// Mitsubishi GX Works2 project: LRI - PLC - A1+Ã1+A2   PLC: Q03UDV

PROGRAM MAIN
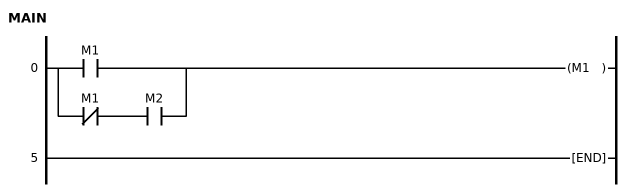
0     LD      M1
      LDI     M1
      AND     M2
      ORB
      OUT     M1
5     END
END_PROGRAM
